Fanuc KAREL source: PROG_RESTORE.kl

PROGRAM T
%NOLOCKGROUP
VAR
 v0 : STRING[40]
 v1 : INTEGER
BEGIN
 PROG_RESTORE(v0, v1)
END T
